FUNCTION_BLOCK Potentiometer (* Composite Function Block Type *)
  (* Standard: 61499-2 *)
  (* Version 0.0, 2011-12-18, 4DIAC-IDE, 4DIAC-Consortium *)
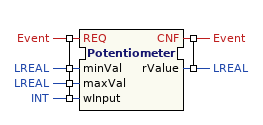
  EVENT_INPUT
    REQ WITH minVal, wInput, maxVal; (* Normal Execution Request *)
  END_EVENT
  EVENT_OUTPUT
    CNF WITH rValue; (* Execution Confirmation *)
  END_EVENT
  VAR_INPUT
    minVal : LREAL; (* Input event qualifier *)
    maxVal : LREAL;
    wInput : INT;
  END_VAR
  VAR_OUTPUT
    rValue : LREAL; (* Output event qualifier *)
  END_VAR
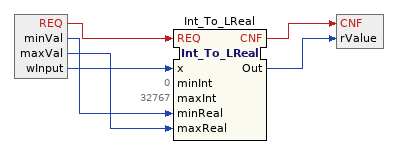
  FBS
    Int_To_LReal : Int_To_LReal(minInt := 0, maxInt := 32767);
  END_FBS
  EVENT_CONNECTIONS
    REQ TO Int_To_LReal.REQ;
    Int_To_LReal.CNF TO CNF;
  END_CONNECTIONS
  DATA_CONNECTIONS
    minVal TO Int_To_LReal.minReal;
    Int_To_LReal.Out TO rValue;
    maxVal TO Int_To_LReal.maxReal;
    wInput TO Int_To_LReal.x;
  END_CONNECTIONS
END_FUNCTION_BLOCK
